Staubli VAL3: QueueFuncs.pjx

--- QueueFuncs.pjx ---
Parameters version=s7.7.2 stackSize=5000 millimeterUnit=true
Program file=clear.pgx
Program file=getNumElems.pgx
Program file=pop.pgx
Program file=push.pgx
Program file=start.pgx
Program file=stop.pgx
Data file=QueueFuncs.dtx
Type name=Queue path=Disk://ros_libs/Queue/Queue.pjx
Type name=MotionCmd path=Disk://ros_libs/MotionCmd/MotionCmd.pjx

--- QueueFuncs.dtx ---


--- start.pgx ---
program start()
begin
end

--- clear.pgx ---
public program clear(Queue& x_qQueue)
begin
  x_qQueue.nElems = 0
  x_qQueue.nPush = x_qQueue.nPop
end

--- getNumElems.pgx ---
public program getNumElems(Queue& x_qQueue, num& x_nNumElems)
begin
  x_nNumElems = x_qQueue.nElems
end

--- pop.pgx ---
public program pop(Queue& x_qQueue, MotionCmd& x_mCmd, bool& x_bRes)
begin
  if (x_qQueue.nElems > 0)
    x_mCmd = x_qQueue.buffer[x_qQueue.nPop]
    x_qQueue.nElems = x_qQueue.nElems - 1
    x_qQueue.nPop = x_qQueue.nPop + 1
    if (x_qQueue.nPop >= size(x_qQueue.buffer))
      x_qQueue.nPop = 0
    endIf
    x_bRes = true
  else
    x_bRes = false
  endIf
end

--- push.pgx ---
public program push(Queue& x_qQueue, MotionCmd& x_mCmd, bool& x_bRes)
begin
  if (x_qQueue.nElems < size(x_qQueue.buffer))
    x_qQueue.buffer[x_qQueue.nPush] = x_mCmd
    x_qQueue.nElems = x_qQueue.nElems + 1
    x_qQueue.nPush = x_qQueue.nPush + 1
    if (x_qQueue.nPush >= size(x_qQueue.buffer))
      x_qQueue.nPush = 0
    endIf
    x_bRes = true
  else
    x_bRes = false
  endIf
end
